{attribute 'qualified_only'}
// Robot8 Data-RightArm
VAR_GLOBAL CONSTANT									 
	// absolute encoder value at minimal joint positon
	g_minLinkEncoder :ARRAY[1..g_mArmNum, 1..g_mJntNum] OF DINT :=
		[122745, 128228, 36292, 22430, 20158, 81422, 0,
		 35855, 68924, 4429, 107164, 130111, 42645, 0];
		 
	// absolute encoder value at maximum joint positon
	g_maxLinkEncoder :ARRAY[1..g_mArmNum, 1..g_mJntNum] OF DINT :=
		[36223, 83720, 69818, 109643, 52927, 61070, 0,
		 79841, 24455, 37956, 63571, 31889, 22283, 0];
	
	// absolute encoder value at calibrated positon
	g_caliLinkEncoder :ARRAY[1..g_mArmNum, 1..g_mJntNum] OF DINT :=
		[13120, 107027, 47903, 76302, 102239, 104240, 53627,
		 57523, 46542, 15769, 8255, 81176, 131007, 56205];
	
	 // if absolute encoder value cross zeros within joint motion range
	 // NOTICE: joint 7 is always 0.
	g_linkEncZeroCross :ARRAY[1..g_mArmNum, 1..g_mJntNum] OF INT :=
		[1, 0, 0, 0, 1, 1, 1,
		 0, 0, 0, 1, 0, 1, 1];
		 
	// limit value of gripper hall sensor
	g_minHallSensorValue :ARRAY[1..2] OF DINT:=[8720383,8982527];
	g_maxHallSensorValue :ARRAY[1..2] OF DINT  :=[95684892,94374153];
		 
 	//################ DO NOT modify parameters below ###########################	
	// abolute encoder expanded limit buffer in case there is calibrtion error at limit position
	g_linkEncLimitBuffer : DINT := 1000;
	
	// flag if joint can rotate multiple cycles
	g_multipleCyclesJoint :ARRAY[1..g_mArmNum, 1..g_mJntNum] OF INT :=
		[0, 0, 0, 0, 0, 0, 1,
		 0, 0, 0, 0, 0, 0, 1];
		 
	// joint position at link encoder calibrated point
	g_linkEncCaliJntPos :ARRAY[1..g_mArmNum, 1..g_mJntNum] OF LREAL :=
		[0.0, -PI/2, 0.0, -pi, pi, -PI/2, 0.0,
		 0.0, -PI/2, 0.0, 0.0, pi, PI/2, 0.0];

END_VAR

(* stored: Version 1.1.0.1, ProductVersion 3.1.4024.12
   GVL GVL_ArmJointCaliData: Id {110f2ddd-8f6e-45b7-a97a-8030310c3113} *)
